FUNCTION_BLOCK FB_SetupArm
VAR_INPUT
END_VAR
VAR_OUTPUT
END_VAR
VAR
	// arm index, from 1 to 4
	m_armIdx: INT;
	
	// joints
	m_joints :ARRAY[1..g_setupJntNum] OF FB_SetupJoint;
	
	// adjust detect
	m_adjustIO AT%I* :UDINT;
	m_manualAdjustOnFlag :BOOL:=FALSE;
	m_jnt5AdjustDir :INT:=0; // -1, 0, 1;
	m_manualAdjustDetect : FB_setupAdjustDetect;
	m_jnt5AdjustDetect : FB_setupJnt5AdjustDetect;
	m_trocarOnFlag :BOOL :=FALSE;
	m_trocarDetect : FB_TrocarDetect;
	
	//arm aseptic cover megnet and  spring breakage from joint 3 check
	m_asepticMegnetSpringBreakCheck  AT %I* :DINT;
	
	// arm cartesian data, defined in cart origin
	m_curCartPose	:ST_Frame;
	
	// cartesion position of remote center
	m_rcPos :Vec3d;	
	
	// arm joint data
	m_curMotorPos :Vec5d;
	m_curLinkPos :Vec5d;
	m_curJntPos :Vec5d;
	m_curJntVel :Vec5d;
	m_curJntTrq :Vec5d;
	m_rawJntCurrent :Vec5d;
	m_filtJntCurrent :Vec5d;
	m_cmdJntCurrent : Vec5d;
	m_cmdJntPos :Vec5d;
	m_cmdJntVel :Vec5d;
	m_cmdJntTrq :Vec5d;
	m_motorEncSalta : vec5di;
	m_lastMotorEnc:Vec5di;
	
	// arm gravity
	m_jntGravity : Vec5d:=g_zeroVec5d;
	m_jntGravityBias :Vec5d :=g_zeroVec5d;
	
	// joint position controller
	m_jntPIDCtrl :ARRAY[1..g_setupJntNum] OF FB_PID;
	
	//arm light out to drive
	m_lightIO AT %Q* :DINT;
	
	// output arm light
	m_SdoWrite:ARRAY [1..4] OF FB_EcCoESdoWrite;
	
	//IP of operating arm
	m_armNetId:T_AmsNetId; 	
	m_setupNetId:T_AmsNetId;
	
	//Joint port number
	m_jointAddrJ3:UINT;	
	m_jointAddrJ8:UINT;	
	m_jointAddrPbox:UINT;
	m_LEDTestCount : UDINT;
	// arm DH 
	m_setupBaseFrame :ST_Frame;
	m_nominalDH:ARRAY[1..5] OF Vec4d;
	m_currentDH:ARRAY[1..5] OF Vec4d;
	
	//check joint 3 spring
	m_dataWrite : BOOL;
	m_dataWriteF : F_TRIG;
	m_jnt3SpringPosInc : LREAL;
	m_jnt3MoveDistance : LREAL;
	m_jnt3MoveDistanceRecord : LREAL;
END_VAR

PROPERTY armIdx : int
GET
armIdx:=m_armIdx;
END_GET
END_PROPERTY

METHOD checkDisplayLED : BOOL
VAR_INPUT
	LEDTestCount : UDINT;
END_VAR


m_LEDTestCount := LEDTestCount;

m_SdoWrite[4](sNetId:= m_setupNetId, nSlaveAddr:= m_jointAddrJ3, nSubIndex:= 06, nIndex:= 16#6090, pSrcBuf:=ADR(m_LEDTestCount) , cbBufLen:=SIZEOF(m_LEDTestCount) , bExecute:= TRUE, tTimeout:= , bBusy=> , bError=> , nErrId=> );
IF NOT m_SdoWrite[4].bBusy THEN
	m_SdoWrite[4](bExecute:=FALSE);
	checkDisplayLED := TRUE;
END_IF
END_METHOD

METHOD PROTECTED checkIO : BOOL
VAR_INPUT
END_VAR
// check manual and auto adjust button
// joint5 and joint1-4 are not allowed to move at the same time 
IF m_manualAdjustOnFlag THEN
	m_manualAdjustOnFlag := m_manualAdjustDetect.run(m_adjustIO);
	m_jnt5AdjustDir:=0;
ELSIF m_jnt5AdjustDir<>0 THEN
	m_jnt5AdjustDir := m_jnt5AdjustDetect.run(m_adjustIO);
	m_manualAdjustOnFlag:=FALSE;
ELSE
	m_manualAdjustOnFlag := m_manualAdjustDetect.run(m_adjustIO);
	m_jnt5AdjustDir := m_jnt5AdjustDetect.run(m_adjustIO);
END_IF

// check trocar
m_trocarOnFlag := m_trocarDetect.run(m_adjustIO);
END_METHOD

METHOD checkLight : BOOL
VAR_INPUT
	i_lightCtrlWord : UDINT;
END_VAR

VAR
	lightCtrlWord : UDINT;
END_VAR
// to PDO
m_lightIO := UDINT_TO_DINT(i_lightCtrlWord);

// trig sdo write
lightCtrlWord := SHL(i_lightCtrlWord,16);
m_SdoWrite[1](sNetId:= m_armNetId, nSlaveAddr:= m_jointAddrJ8, nSubIndex:= 0, nIndex:= 16#6092, pSrcBuf:=ADR(lightCtrlWord) , cbBufLen:=SIZEOF(lightCtrlWord) , bExecute:= TRUE, tTimeout:= , bBusy=> , bError=> , nErrId=> );
m_SdoWrite[2](sNetId:= m_armNetId, nSlaveAddr:= m_jointAddrJ3, nSubIndex:= 0, nIndex:= 16#6092, pSrcBuf:=ADR(lightCtrlWord) , cbBufLen:=SIZEOF(lightCtrlWord) , bExecute:= TRUE, tTimeout:= , bBusy=> , bError=> , nErrId=> );
m_SdoWrite[3](sNetId:= m_armNetId, nSlaveAddr:= m_jointAddrPbox, nSubIndex:= 0, nIndex:= 16#6092, pSrcBuf:= ADR(lightCtrlWord), cbBufLen:= SIZEOF(lightCtrlWord), bExecute:= TRUE, tTimeout:= , bBusy=> , bError=> , nErrId=> );

// disable sdo write
IF NOT m_SdoWrite[1].bBusy AND  NOT m_SdoWrite[2].bBusy THEN
	m_SdoWrite[1](bExecute:=FALSE);
	m_SdoWrite[2](bExecute:=FALSE);
	m_SdoWrite[3](bExecute:=FALSE);
END_IF
END_METHOD

METHOD checkSpring : BOOL
VAR_INPUT
END_VAR
//joint 3 spring movement distance
IF  m_joints[3].isEnabled() THEN
	m_jnt3SpringPosInc := m_jnt3SpringPosInc +  ABS(m_curJntVel[3] * g_setupArmCtrlCycleTime);
	m_jnt3MoveDistance := m_jnt3MoveDistanceRecord + m_jnt3SpringPosInc;
END_IF
m_dataWriteF(CLK:= m_joints[3].isEnabled(), Q=> m_dataWrite);
IF m_dataWrite THEN
	m_jnt3MoveDistanceRecord := m_jnt3MoveDistance;
	m_jnt3SpringPosInc := 0;
	m_dataWrite := FALSE;
END_IF
END_METHOD

PROPERTY cmdJntCurrent : REFERENCE TO  Vec5d
GET
cmdJntCurrent ref= m_cmdJntCurrent;
END_GET
END_PROPERTY

PROPERTY curCartPose : REFERENCE TO ST_Frame
GET
curCartPose ref=m_curCartPose;
END_GET
END_PROPERTY

PROPERTY curJntPos : REFERENCE TO Vec5d
GET
curJntPos ref=m_curJntPos;
END_GET
END_PROPERTY

PROPERTY curJntTrq : REFERENCE TO Vec5d
GET
curJntTrq ref=m_curJntTrq;
END_GET
END_PROPERTY

PROPERTY curJntVel :REFERENCE TO Vec5d
GET
curJntVel ref=m_curJntVel;
END_GET
END_PROPERTY

PROPERTY curLinkPos :REFERENCE TO Vec5d
GET
curLinkPos ref=m_curLinkPos;
END_GET
END_PROPERTY

PROPERTY curMotorPos : REFERENCE TO  Vec5d
GET
curMotorPos ref=m_curMotorPos;
END_GET
END_PROPERTY

METHOD PUBLIC enable : BOOL
VAR_IN_OUT CONSTANT
	i_jntIdx :Vec5i;
END_VAR
VAR
	i :INT ;
END_VAR
FOR i:=1 TO g_setupJntNum DO
	IF 1= i_jntIdx[i] THEN
		m_joints[i].enable();
	ELSE
		m_joints[i].disable();
	END_IF
END_FOR
END_METHOD

PROPERTY filtJntCurrent :REFERENCE TO Vec5d
GET
filtJntCurrent ref= m_filtJntCurrent;
END_GET
END_PROPERTY

// compute cartesion pose in cart origin
METHOD PROTECTED forwardKinematic : BOOL
VAR_IN_OUT CONSTANT
	i_jntPos :Vec5d;
END_VAR
VAR_IN_OUT
	r_cartPose :ST_Frame;
	
	// position of remote center
	r_rcPos :Vec3d;
END_VAR
VAR
	cf1,cf2,cf3,cf4,c1,c2,c3,c4,c5 :LREAL;
	sf1,sf2,sf3,sf4,s1,s2,s3,s4,s5 :LREAL;
	a1,a2 :LREAL;
	d1,d2,d3:LREAL;
	
	s1c2, s12, c12, c1s2,  sf12, sf1cf2, cf1sf2, cf12, sf23, sf2cf3, cf23, cf2sf3:LREAL;
	c1s2cf1, cf1s1c2, c3s2sf1, s2s3sf1, c1sf1cf2,c12cf1, c2sf12,s1sf12,c2sf1cf2,c1sf12,s1sf1cf2,cf1s12 :LREAL;
	
	posVec1, posVec2:Vec3d;
	fixPointMatrix:ARRAY[1..4,1..4] OF LREAL;
END_VAR
a1:=m_nominalDH[2][2];
a2:=m_nominalDH[5][2];

d1:=m_nominalDH[2][4]+i_jntPos[2];
d2:=m_nominalDH[3][4]+i_jntPos[3];
d3:=m_nominalDH[5][4];

cf1:=COS(m_nominalDH[2][1]);
cf2:=COS(m_nominalDH[3][1]);
cf3:=COS(m_nominalDH[4][1]);
cf4:=COS(m_nominalDH[5][1]);
c1:=COS(m_nominalDH[1][3]+i_jntPos[1]);
c2:=COS(m_nominalDH[2][3]);
c3:=COS(m_nominalDH[3][3]);
c4:=COS(m_nominalDH[4][3]+i_jntPos[4]);
c5:=COS(m_nominalDH[5][3]+i_jntPos[5]);


sf1:=SIN(m_nominalDH[2][1]);
sf2:=SIN(m_nominalDH[3][1]);
sf3:=SIN(m_nominalDH[4][1]);
sf4:=SIN(m_nominalDH[5][1]);
s1:=SIN(m_nominalDH[1][3]+i_jntPos[1]);
s2:=SIN(m_nominalDH[2][3]);
s3:=SIN(m_nominalDH[3][3]);
s4:=SIN(m_nominalDH[4][3]+i_jntPos[4]);
s5:=SIN(m_nominalDH[5][3]+i_jntPos[5]);

s1c2:=s1*c2;
s12:=s1*s2;
c12:=c1*c2;
c1s2:=c1*s2;
sf12:=sf1*sf2;
sf1cf2:=sf1*cf2;
cf12:=cf1*cf2;
cf1sf2:=cf1*sf2;
sf2cf3:=sf2*cf3;
sf23:=sf2*sf3;
cf23:=cf2*cf3;
cf2sf3:=cf2*sf3;
c1s2cf1:=c1s2*cf1;
cf1s1c2:=cf1*s1c2;
c3s2sf1:=c3*s2*sf1;
s2s3sf1:=s2*s3*sf1;
c1sf1cf2:=c1*sf1cf2;
c12cf1:=c12*cf1;
c2sf12:=c2*sf12;
s1sf12:=s1*sf12;
c2sf1cf2:=c2*sf1cf2;
c1sf12:=c1*sf12;
s1sf1cf2:=s1*sf1cf2;
cf1s12:=cf1*s12;

r_cartPose.m_pos[1]:=a1*c1 + d2*(s1sf1cf2 + sf2*(c1s2 + cf1s1c2)) - d3*(cf4*(sf3*(c3*(s1sf12 - cf2*(c1s2 + cf1s1c2)) - s3*(c12 - cf1s12)) - cf3*(s1sf1cf2 + sf2*(c1s2 + cf1s1c2))) - sf4*(s4*(s3*(s1sf12 - cf2*(c1s2 + cf1s1c2)) 
					+ c3*(c12 - cf1s12)) - c4*(cf3*(c3*(s1sf12 - cf2*(c1s2 + cf1s1c2)) - s3*(c12 - cf1s12)) + sf3*(s1sf1cf2 + sf2*(c1s2 + cf1s1c2))))) + a2*(c4*(s3*(s1sf12 - cf2*(c1s2 + cf1s1c2)) + c3*(c12 - cf1s12)) 
					+ s4*(cf3*(c3*(s1sf12 - cf2*(c1s2 + cf1s1c2)) - s3*(c12 - cf1s12)) + sf3*(s1sf1cf2 + sf2*(c1s2 + cf1s1c2)))) + d1*s1*sf1; 
r_cartPose.m_pos[2]:=d3*(cf4*(sf3*(c3*(c1sf12 + cf2*(s12 - c12cf1)) + s3*(s1c2 + c1s2cf1)) - cf3*(c1sf1cf2 - sf2*(s12 - c12cf1))) - sf4*(s4*(s3*(c1sf12 + cf2*(s12 - c12cf1)) - c3*(s1c2 + c1s2cf1)) - c4*(sf3*(c1sf1cf2 - sf2*(s12 - c12cf1)) 
					+ cf3*(c3*(c1sf12 + cf2*(s12 - c12cf1)) + s3*(s1c2 + c1s2cf1))))) - d2*(c1sf1cf2 - sf2*(s12 - c12cf1)) + a1*s1 - a2*(s4*(sf3*(c1sf1cf2 - sf2*(s12 - c12cf1)) + cf3*(c3*(c1sf12 + cf2*(s12 - c12cf1)) + s3*(s1c2 + c1s2cf1))) 
					+ c4*(s3*(c1sf12 + cf2*(s12 - c12cf1)) - c3*(s1c2 + c1s2cf1))) - c1*d1*sf1; 
r_cartPose.m_pos[3]:=cf1*d1 - d3*(sf4*(c4*(cf3*(c3*(cf1sf2 + c2sf1cf2) - s2s3sf1) + sf3*(cf12 - c2sf12)) - s4*(s3*(cf1sf2 + c2sf1cf2) + c3s2sf1)) + cf4*(sf3*(c3*(cf1sf2 + c2sf1cf2) - s2s3sf1) - cf3*(cf12 - c2sf12))) 
					+ a2*(s4*(cf3*(c3*(cf1sf2 + c2sf1cf2) - s2s3sf1) + sf3*(cf12 - c2sf12)) + c4*(s3*(cf1sf2 + c2sf1cf2) + c3s2sf1)) + d2*(cf12 - c2sf12);

r_cartPose.m_rot[1,1]:=c5*(c4*(s3*(s1sf12 - cf2*(c1s2 + cf1s1c2)) + c3*(c12 - cf1s12)) + s4*(cf3*(c3*(s1sf12 - cf2*(c1s2 + cf1s1c2)) - s3*(c12 - cf1s12)) + sf3*(s1sf1cf2 + sf2*(c1s2 + cf1s1c2)))) - s5*(sf4*(sf3*(c3*(s1sf12 - cf2*(c1s2 + cf1s1c2))
					 - s3*(c12 - cf1s12)) - cf3*(s1sf1cf2 + sf2*(c1s2 + cf1s1c2))) + cf4*(s4*(s3*(s1sf12 - cf2*(c1s2 + cf1s1c2)) + c3*(c12 - cf1s12)) - c4*(cf3*(c3*(s1sf12 - cf2*(c1s2 + cf1s1c2)) - s3*(c12 - cf1s12)) + sf3*(s1sf1cf2 + sf2*(c1s2 + cf1s1c2)))));  
r_cartPose.m_rot[1,2]:=- c5*(sf4*(sf3*(c3*(s1sf12 - cf2*(c1s2 + cf1s1c2)) - s3*(c12 - cf1s12)) - cf3*(s1sf1cf2 + sf2*(c1s2 + cf1s1c2))) + cf4*(s4*(s3*(s1sf12 - cf2*(c1s2 + cf1s1c2)) + c3*(c12 - cf1s12)) - c4*(cf3*(c3*(s1sf12 - cf2*(c1s2 + cf1s1c2))
					 - s3*(c12 - cf1s12)) + sf3*(s1sf1cf2 + sf2*(c1s2 + cf1s1c2))))) - s5*(c4*(s3*(s1sf12 - cf2*(c1s2 + cf1s1c2)) + c3*(c12 - cf1s12)) + s4*(cf3*(c3*(s1sf12 - cf2*(c1s2 + cf1s1c2)) - s3*(c12 - cf1s12)) + sf3*(s1sf1cf2 + sf2*(c1s2 + cf1s1c2))));  
r_cartPose.m_rot[1,3]:=sf4*(s4*(s3*(s1sf12 - cf2*(c1s2 + cf1s1c2)) + c3*(c12 - cf1s12)) - c4*(cf3*(c3*(s1sf12 - cf2*(c1s2 + cf1s1c2)) - s3*(c12 - cf1s12)) + sf3*(s1sf1cf2 + sf2*(c1s2 + cf1s1c2)))) - cf4*(sf3*(c3*(s1sf12 - cf2*(c1s2 + cf1s1c2))
					 - s3*(c12 - cf1s12)) - cf3*(s1sf1cf2 + sf2*(c1s2 + cf1s1c2)));
r_cartPose.m_rot[2,1]:=s5*(sf4*(sf3*(c3*(c1sf12 + cf2*(s12 - c12cf1)) + s3*(s1c2 + c1s2cf1)) - cf3*(c1sf1cf2 - sf2*(s12 - c12cf1))) + cf4*(s4*(s3*(c1sf12 + cf2*(s12 - c12cf1)) - c3*(s1c2 + c1s2cf1)) - c4*(sf3*(c1sf1cf2 - sf2*(s12 - c12cf1))
					 + cf3*(c3*(c1sf12 + cf2*(s12 - c12cf1)) + s3*(s1c2 + c1s2cf1))))) - c5*(s4*(sf3*(c1sf1cf2 - sf2*(s12 - c12cf1)) + cf3*(c3*(c1sf12 + cf2*(s12 - c12cf1)) + s3*(s1c2 + c1s2cf1))) + c4*(s3*(c1sf12 + cf2*(s12 - c12cf1))
					 - c3*(s1c2 + c1s2cf1))); 
r_cartPose.m_rot[2,2]:=c5*(sf4*(sf3*(c3*(c1sf12 + cf2*(s12 - c12cf1)) + s3*(s1c2 + c1s2cf1)) - cf3*(c1sf1cf2 - sf2*(s12 - c12cf1))) + cf4*(s4*(s3*(c1sf12 + cf2*(s12 - c12cf1)) - c3*(s1c2 + c1s2cf1)) - c4*(sf3*(c1sf1cf2 - sf2*(s12 - c12cf1))
					+ cf3*(c3*(c1sf12 + cf2*(s12 - c12cf1)) + s3*(s1c2 + c1s2cf1))))) + s5*(s4*(sf3*(c1sf1cf2 - sf2*(s12 - c12cf1)) + cf3*(c3*(c1sf12 + cf2*(s12 - c12cf1)) + s3*(s1c2 + c1s2cf1))) + c4*(s3*(c1sf12 + cf2*(s12 - c12cf1))
					 - c3*(s1c2 + c1s2cf1)));  
r_cartPose.m_rot[2,3]:=cf4*(sf3*(c3*(c1sf12 + cf2*(s12 - c12cf1)) + s3*(s1c2 + c1s2cf1)) - cf3*(c1sf1cf2 - sf2*(s12 - c12cf1))) - sf4*(s4*(s3*(c1sf12 + cf2*(s12 - c12cf1)) - c3*(s1c2 + c1s2cf1)) - c4*(sf3*(c1sf1cf2 - sf2*(s12 - c12cf1)) 
					+ cf3*(c3*(c1sf12 + cf2*(s12 - c12cf1)) + s3*(s1c2 + c1s2cf1))));
r_cartPose.m_rot[3,1]:=s5*(cf4*(c4*(cf3*(c3*(cf1sf2 + c2sf1cf2) - s2s3sf1) + sf3*(cf12 - c2sf12)) - s4*(s3*(cf1sf2 + c2sf1cf2) + c3s2sf1)) - sf4*(sf3*(c3*(cf1sf2 + c2sf1cf2) - s2s3sf1) - cf3*(cf12 - c2sf12))) + c5*(s4*(cf3*(c3*(cf1sf2 + c2sf1cf2)
					 - s2s3sf1) + sf3*(cf12 - c2sf12)) + c4*(s3*(cf1sf2 + c2sf1cf2) + c3s2sf1));  
r_cartPose.m_rot[3,2]:=c5*(cf4*(c4*(cf3*(c3*(cf1sf2 + c2sf1cf2) - s2s3sf1) + sf3*(cf12 - c2sf12)) - s4*(s3*(cf1sf2 + c2sf1cf2) + c3s2sf1)) - sf4*(sf3*(c3*(cf1sf2 + c2sf1cf2) - s2s3sf1) - cf3*(cf12 - c2sf12))) - s5*(s4*(cf3*(c3*(cf1sf2 + c2sf1cf2)
					 - s2s3sf1) + sf3*(cf12 - c2sf12)) + c4*(s3*(cf1sf2 + c2sf1cf2) + c3s2sf1));  
r_cartPose.m_rot[3,3]:=- sf4*(c4*(cf3*(c3*(cf1sf2 + c2sf1cf2) - s2s3sf1) + sf3*(cf12 - c2sf12)) - s4*(s3*(cf1sf2 + c2sf1cf2) + c3s2sf1)) - cf4*(sf3*(c3*(cf1sf2 + c2sf1cf2) - s2s3sf1) - cf3*(cf12 - c2sf12));

r_cartPose:=transform(m_setupBaseFrame, r_cartPose);
//********************output2:remote center position************************//
posVec1[1]:=0;
posVec1[2]:=-GVL_SlaveArmKinematic.g_d1;
posVec1[3]:=0;
matMultiVec(r_cartPose.m_rot, posVec1,posVec2);
vecAdd(r_cartPose.m_pos,posVec2, posVec1);
r_rcPos:=posVec1;
END_METHOD

METHOD PUBLIC init : BOOL
VAR_INPUT
	i_armIdx:INT;
END_VAR
VAR 
	i :INT ;
	currentRatioMotor2Jnt:LREAL;
END_VAR
// arm statues init
m_armIdx:=i_armIdx;

// arm DH
initDH();

// joint init
FOR i:=1 TO g_setupJntNum DO
	m_joints[i].init(m_armIdx, i,g_setupArmCtrlCycleTime);
END_FOR

// joint init
FOR i:=1 TO g_setupJntNum DO
	m_joints[i].initJntPos();
END_FOR

// update arm status if joint position is re-init
updateStatus();

// joint controller init
FOR i:=1 TO g_setupJntNum DO 
	currentRatioMotor2Jnt:=GVL_SetupMotorParameters.g_motorTrqConst[i]*GVL_SetupMotorParameters.g_motorReduction[i]/1000;
	m_jntPIDCtrl[i].init(g_setupArmCtrlCycleTime,GVL_SetupControlParameters.g_posKp[i],GVL_SetupControlParameters.g_posKd[i],
		GVL_SetupControlParameters.g_posKi[i], GVL_SetupControlParameters.g_posKiLimit[i]* currentRatioMotor2Jnt,
		GVL_SetupControlParameters.g_posCtrlLimit[i]*currentRatioMotor2Jnt);
END_FOR

//init arm netID and adrr
m_armNetId := GVL_SystemParameters.g_slaveArmNetID[armIdx];
m_jointAddrJ3 := GVL_SystemParameters.g_setupJointNetPort[armIdx,3];
m_jointAddrJ8 := GVL_SystemParameters.g_slaveJointNetPort[armIdx,3];
m_jointAddrPbox := GVL_SystemParameters.g_slaveJointNetPort[armIdx,4];

//joint 3 spring check
m_jnt3MoveDistance := m_jnt3MoveDistanceRecord;
END_METHOD

METHOD initDH : BOOL
VAR_INPUT
END_VAR
VAR
	i,j :INT;
	DHErr:ARRAY[1..8,1..4] OF LREAL;
END_VAR
// DH error
IF (m_armIdx=1) THEN
	DHErr := GVL_SlaveArmKinematic.g_slaveArm1DHErr;
	FOR i:=1 TO 3 DO
		FOR j:=1 TO 3 DO 
			m_setupBaseFrame.m_rot[i,j]:= GVL_SlaveArmKinematic.g_slaveArm1Base[i,j];
		END_FOR
		m_setupBaseFrame.m_pos[i]:= GVL_SlaveArmKinematic.g_slaveArm1Base[i,4];
	END_FOR
	
ELSIF (m_armIdx=2) THEN
	DHErr := GVL_SlaveArmKinematic.g_slaveArm2DHErr;
	FOR i:=1 TO 3 DO
		FOR j:=1 TO 3 DO 
			m_setupBaseFrame.m_rot[i,j]:= GVL_SlaveArmKinematic.g_slaveArm2Base[i,j];
		END_FOR
		m_setupBaseFrame.m_pos[i]:= GVL_SlaveArmKinematic.g_slaveArm2Base[i,4];
	END_FOR
	
ELSIF (m_armIdx=3) THEN	
	DHErr := GVL_SlaveArmKinematic.g_slaveArm3DHErr;
	FOR i:=1 TO 3 DO
		FOR j:=1 TO 3 DO 
			m_setupBaseFrame.m_rot[i,j]:= GVL_SlaveArmKinematic.g_slaveArm3Base[i,j];
		END_FOR
		m_setupBaseFrame.m_pos[i]:= GVL_SlaveArmKinematic.g_slaveArm3Base[i,4];
	END_FOR
	
ELSIF (m_armIdx=4) THEN	
	DHErr := GVL_SlaveArmKinematic.g_slaveArm4DHErr;
	FOR i:=1 TO 3 DO
		FOR j:=1 TO 3 DO 
			m_setupBaseFrame.m_rot[i,j]:= GVL_SlaveArmKinematic.g_slaveArm4Base[i,j];
		END_FOR
		m_setupBaseFrame.m_pos[i]:= GVL_SlaveArmKinematic.g_slaveArm4Base[i,4];
	END_FOR
END_IF

FOR i:=1 TO 5 DO 
	FOR j:=1 TO 4 DO
		m_nominalDH[i][j]:= GVL_SetupArmKinematic.g_setupArmDH[i,j] + DHErr[i,j];
	END_FOR	
END_FOR
m_nominalDH[2][2]:= GVL_SetupArmKinematic.g_setupA2[m_armIdx] + DHErr[2,2];
m_nominalDH[3][4]:= GVL_SetupArmKinematic.g_setupD4[m_armIdx] + DHErr[3,4];
END_METHOD

METHOD PUBLIC isEnabled : BOOL
VAR_IN_OUT CONSTANT
	i_jntIdx :Vec5i;
END_VAR
VAR
	i :INT ;
END_VAR
isEnabled := TRUE;
FOR i:=1 TO g_setupJntNum DO
	IF 1= i_jntIdx[i] THEN
		isEnabled :=  (m_joints[i].isEnabled() AND isEnabled);
	END_IF
END_FOR
END_METHOD

PROPERTY jnt5AdjustDir : int
GET
jnt5AdjustDir := m_jnt5AdjustDir;
END_GET
END_PROPERTY

PROPERTY jntGravity :REFERENCE TO Vec5d
GET
jntGravity ref=m_jntGravity;
END_GET
END_PROPERTY

PROPERTY jntGravityBias :REFERENCE to Vec5d
GET
jntGravityBias ref=m_jntGravityBias;
END_GET
SET // PUBLIC
m_jntGravityBias := jntGravityBias;
END_SET
END_PROPERTY

PROPERTY manualAdjustOn : bool
GET
manualAdjustOn := m_manualAdjustOnFlag;
END_GET
END_PROPERTY

PROPERTY motorEncSalta : REFERENCE TO Vec5di
GET
motorEncSalta ref= m_motorEncSalta;
END_GET
END_PROPERTY

PROPERTY rawJntCurrent :REFERENCE TO Vec5d
GET
rawJntCurrent ref=m_rawJntCurrent;
END_GET
END_PROPERTY

PROPERTY rcPos :REFERENCE to Vec3d
GET
rcPos REF= m_rcPos;
END_GET
END_PROPERTY

PROPERTY PUBLIC trocarOn : bool
GET
trocarOn := m_trocarOnFlag;
END_GET
END_PROPERTY

// update joints control command
METHOD PUBLIC updateCmds : BOOL
VAR_IN_OUT CONSTANT
	i_armCtrlCmd : ST_SetupArmCtrlCmds;
END_VAR
VAR
	i:INT;
END_VAR
m_cmdJntTrq:=i_armCtrlCmd.m_cmdJntTrq;
m_cmdJntPos :=i_armCtrlCmd.m_cmdJntPos;
m_cmdJntVel :=i_armCtrlCmd.m_cmdJntVel;

// enable/disable joints
enable(i_armCtrlCmd.m_jntEnableFlag);

// position/torque control
FOR i:=1 TO g_setupJntNum DO 
	IF i_armCtrlCmd.m_jntOPMode[i]=DriverOPMode_PosTrq THEN
		// position controller and gravity feedforward
		m_cmdJntTrq[i]:=m_jntPIDCtrl[i].run(m_cmdJntPos[i],m_curJntPos[i],0,m_curJntVel[i]);
		m_cmdJntTrq[i]:=m_cmdJntTrq[i]+m_jntGravity[i];
		m_joints[i].updateCmds(DriverOPMode_Trq,m_cmdJntPos[i],m_cmdJntTrq[i]);
	ELSIF i_armCtrlCmd.m_jntOPMode[i]=DriverOPMode_Trq THEN
		// gravity feedforward
		m_jntPIDCtrl[i].reset();
		m_cmdJntTrq[i]:=m_cmdJntTrq[i]+m_jntGravity[i]+m_jntGravityBias[i]+GVL_SetupArmDynamics.g_setupJntGravityOffset[m_armIdx, i];
		m_joints[i].updateCmds(DriverOPMode_Trq,i_armCtrlCmd.m_cmdJntPos[i],m_cmdJntTrq[i]);
	ELSE
		m_jntPIDCtrl[i].reset();
		m_cmdJntTrq[i]:=0;
		m_joints[i].updateCmds(DriverOPMode_Pos,i_armCtrlCmd.m_cmdJntPos[i],m_cmdJntTrq[i]);
	END_IF
	
END_FOR
END_METHOD

METHOD PUBLIC updateDyna : BOOL
VAR_IN_out constant
	i_jnt3Gravity :LREAL;
	i_jnt5Gravity :LREAL;
END_VAR
m_jntGravity[3]:=i_jnt3Gravity;
m_jntGravity[5]:=i_jnt5Gravity;
END_METHOD

// update arm status, including kinematic and dynamic
METHOD PUBLIC updateStatus : BOOL
VAR_INPUT
END_VAR
VAR 
	i,j:INT;
END_VAR
// update joint data
FOR i:=1 TO g_setupJntNum DO
	m_joints[i].updateStatus();
END_FOR

// check adjust button
checkIO();

// get joint data
FOR i:=1 TO g_setupJntNum DO
	m_curMotorPos[i]:=m_joints[i].motorPos;
	m_curLinkPos[i]:=m_joints[i].linkPos;
	m_curJntPos[i]:=m_joints[i].jntPos;
	m_curJntVel[i]:=m_joints[i].jntVel;
	m_curJntTrq[i]:=m_joints[i].jntTrq;
	m_rawJntCurrent[i]:=m_joints[i].rawCurrent;
	m_filtJntCurrent[i]:=m_joints[i].filtCurrent;
	m_cmdJntCurrent[i]:=m_joints[i].cmdCurrent;
	m_motorEncSalta[i] := ABS(m_joints[i].m_motorInputs.m_motorEncoder - m_lastMotorEnc[i]);
	m_lastMotorEnc[i] := m_joints[i].m_motorInputs.m_motorEncoder;
END_FOR 

//check joint 3 spring
checkSpring();

// cartesion pose
forwardKinematic(m_curJntPos,m_curCartPose,m_rcPos);
END_METHOD

END_FUNCTION_BLOCK

(* stored: Version 1.1.0.1, ProductVersion 3.1.4024.11
   POU FB_SetupArm: Id {5c9438f2-768b-4fff-9bfc-3693d995bd67}, SpecialFunc None
   Folder property: Id {c6ea0166-9703-475a-8e8e-3d0d51737a97}
   Property armIdx: Id {cabfa044-e4b7-4d76-b1b7-570e090205fc}
   Get Get: Id {5a987e19-0654-4dd3-bef9-5cc1d433e846}
   Method checkDisplayLED: Id {da0d522c-94f4-492f-8290-51c3f54d3805}
   Method checkIO: Id {fbd89c1b-d255-40db-a7aa-cd2a052b5167}
   Method checkLight: Id {bd15e90e-7362-4cca-a66a-2b7a8c5d2239}
   Method checkSpring: Id {94e88eb3-5f4c-41b2-a2f4-be0ea6fbdbc7}
   Property cmdJntCurrent: Id {cf988543-58f5-435a-b7be-8f2740b3e7a6}
   Get Get: Id {00d8453b-1f45-4430-a6c7-bf4d2acc9ee1}
   Property curCartPose: Id {8b2d212c-f874-4df3-89c4-7a4c59a2497a}
   Get Get: Id {bff86ca2-da06-43d9-9418-b85d681657e9}
   Property curJntPos: Id {dce3bb79-9314-492e-9e98-fee04b74bd41}
   Get Get: Id {f8fadb86-6639-4fb2-a004-3b9df6fdd326}
   Property curJntTrq: Id {24ed19ef-7464-464e-880d-ef73a35a91a7}
   Get Get: Id {1774936a-ec78-4224-9f8a-11723c469020}
   Property curJntVel: Id {9c9eaed8-cbbc-4877-ac64-499b2f94549f}
   Get Get: Id {b341161a-d6a1-4f46-b87e-cd6dfc707fcd}
   Property curLinkPos: Id {31801798-9071-4878-9aba-12be0ad3e45d}
   Get Get: Id {246fe2c5-593e-4bd7-9156-a5d90d9026f6}
   Property curMotorPos: Id {2f4e185f-8286-482d-a2ae-9905a1d92411}
   Get Get: Id {970d1fb2-cdea-4a61-a53b-2160ac80684b}
   Method enable: Id {de5f38b7-8c95-4013-a120-bc96550e0d76}
   Property filtJntCurrent: Id {4315db90-bd10-4e4f-ab74-b8b2244311b8}
   Get Get: Id {9c348772-1b97-4208-9443-80c5fa591884}
   Method forwardKinematic: Id {49767c62-0ec4-4ada-b054-e0d81ad3f08d}
   Method init: Id {38d8d9c7-7db7-4b7f-9fc0-1defdd94f779}
   Method initDH: Id {0377fdc1-4f97-4933-87ed-40408946246d}
   Method isEnabled: Id {b985692a-f6f7-460a-be8e-c41aacfdf6d5}
   Property jnt5AdjustDir: Id {9c383f15-8b4b-4f35-9c30-cbfe61f1e499}
   Get Get: Id {cda39ef3-97eb-493e-a5be-521a72a7dc1b}
   Property jntGravity: Id {33c6cc0e-6d37-4855-b1be-0f076b081ccc}
   Get Get: Id {676c5d39-ab4d-45da-b342-fb30a86742c9}
   Property jntGravityBias: Id {98e9447b-dbcb-43f9-9939-c5f9658d66f6}
   Get Get: Id {45c5ec0b-01e0-48e0-8f64-7a1d89f2d1fe}
   Set Set: Id {4abadf39-71db-4fe9-89b5-4fa9c3a50b80}
   Property manualAdjustOn: Id {06fd6985-ca41-4e66-8b96-f30c8a6d0e2c}
   Get Get: Id {6b9e44f9-af7c-4368-b8c0-d50cceeb95b2}
   Property motorEncSalta: Id {2d50a2e5-10e1-40ef-89d8-499621d72a5e}
   Get Get: Id {b34f3e43-76a6-4223-b561-daf4a431df16}
   Property rawJntCurrent: Id {55d5ae20-b171-429a-ac31-06e15bf272af}
   Get Get: Id {6e301cc8-e411-4dac-b4d8-a08e42ea0f2d}
   Property rcPos: Id {3ac624a0-ed54-4971-a738-0ad5e73415ba}
   Get Get: Id {e3e500a4-2327-4159-bdc5-53a60fab73a3}
   Property trocarOn: Id {1f7ffdba-b6f7-4752-8981-43bd23a041b0}
   Get Get: Id {5ea85821-1b7c-464a-945d-cbdff065bbdf}
   Method updateCmds: Id {6d34fc6a-e3f4-42a7-8c5b-e82cddc386d1}
   Method updateDyna: Id {f00121ef-1617-4216-ab61-3a405eda46ec}
   Method updateStatus: Id {bb24dca5-7706-495a-abc4-658f70a32369} *)
